FUNCTION_BLOCK ItpResetFastMFuncEx
VAR_INPUT
	bExecute:	BOOL;
	nMFuncNo:	UINT;
	tTimeOut:	TIME := DEFAULT_ADS_TIMEOUT;
END_VAR
VAR_IN_OUT
	sNciToPlc:	NciChannelToPlc;
END_VAR
VAR_OUTPUT
	bBusy:	BOOL	:= FALSE;
	bErr:		BOOL	:= FALSE;
	nErrId:	UDINT	:= 0;
END_VAR
VAR
	nState:		UDINT := 0;
	fbItpResetFastMFunc:	ItpResetFastMFunc;
END_VAR
CASE nState OF
0:
	IF bExecute THEN
		IF ItpGetItfVersion( sNciToPlc ) > 0 THEN
			fbItpResetFastMFunc(
				bExecute	:= TRUE,
				nChnId	:= ItpGetChannelId( sNciToPlc ),
				nMFuncNo	:= nMFuncNo,
				tTimeOut:= tTimeOut,
				bBusy	=> bBusy,
				bErr	=> bErr,
				nErrId=> nErrId );
			nState	:= 10;
		ELSE
			bBusy		:= TRUE;
			bErr		:= TRUE;
			nErrId	:= ErrTcNciItp_ItfVersion;
			nState	:= 9999;
		END_IF
	END_IF
10:
	fbItpResetFastMFunc();
	IF NOT fbItpResetFastMFunc.bBusy THEN
		bBusy	:= FALSE;
		IF NOT fbItpResetFastMFunc.bErr THEN
			IF NOT bExecute THEN
				fbItpResetFastMFunc( bExecute := FALSE );
				nState	:= 0;
			ELSE
				nState	:= 9999;
			END_IF
		ELSE
			bErr		:= TRUE;
			nErrId	:= fbItpResetFastMFunc.nErrId;
			nState	:= 9999;
		END_IF
	END_IF

9999:
	fbItpResetFastMFunc( bExecute:=FALSE );
	bBusy	:= FALSE;
	IF NOT bExecute THEN
		nState	:= 0;
	END_IF

END_CASE
END_FUNCTION_BLOCK

(* POU ItpRetraceMoveBackward, ST *)
(*==========================================================*)
(* Name:			ItpRetraceMoveBackward  							*)
(* Desc:			THIS IS NOT A RELEASED IMPLEMENTATION AND    *)
(*             SUBJECT TO CHANGE                            *)
(*             Moving backward                              *)
(*             - program stopped with ItpEStop              *)
(*             - FeederBackup must be enabled               *)
(* Author:	 	kbn														*)
(* Date:			07-december-2006										*)
(* last edit:	VER 6.2.33 						                  *)
(*==========================================================*)
FUNCTION_BLOCK ItpRetraceMoveBackward
VAR_INPUT
	bExecute:	BOOL;
	tTimeOut:	TIME := DEFAULT_ADS_TIMEOUT;
END_VAR
VAR_IN_OUT
	sNciToPlc:	NciChannelToPlc;
END_VAR
VAR_OUTPUT
	bBusy:		BOOL	:= FALSE;
	bErr:			BOOL	:= FALSE;
	nErrId:		UDINT	:= 0;
END_VAR
VAR
	nState:		UDINT	:= 0;
	nData:		UDINT	:= 0;
	fbAdsWrite:	ADSWRITE;
	tDummy:		ST_ItpRetrace;
	fbIsBackupEnabled:ItpIsFeederBackupEnabled;
END_VAR
CASE nState OF
0:
	IF bExecute THEN
		IF ItpGetItfVersion( sNciToPlc ) >= 3 THEN
			bBusy		:= TRUE;
			bErr		:= FALSE;
			nErrId	:= 0;
			nState	:= 10;
		ELSE
			bBusy		:= TRUE;
			bErr		:= TRUE;
			nErrId	:= ErrTcNciItp_ItfVersion;
			nState	:= 9999;
		END_IF
	END_IF
10:
	(* check, if backup is enabled *)
	fbIsBackupEnabled(
		bExecute	:= TRUE,
		tTimeOut	:= tTimeOut,
		sNciToPlc:= sNciToPlc );
	IF NOT fbIsBackupEnabled.bBusy THEN
		IF NOT fbIsBackupEnabled.bErr THEN
			IF fbIsBackupEnabled.bEnabled THEN
				nState	:= 15;
			ELSE
				(* not enabled - fire an error *)
				bErr		:= TRUE;
				nErrId	:= ErrTcNciItp_NotEnabled;
				nState	:= 9999;
			END_IF
		ELSE
			bErr		:= TRUE;
			nErrId	:= fbIsBackupEnabled.nErrId;
			nState	:= 9999;
		END_IF
		fbIsBackupEnabled( bExecute := FALSE, sNciToPlc:= sNciToPlc );
	END_IF

15:
	(* add some code to ensure, that axes stand still *)
	(* in the moment I just check, if e-stop is active *)
	IF NOT ItpIsEStopEx( sNciToPlc ) THEN
		bErr		:= TRUE;
		nErrId	:= ErrTcNciItp_NotReady;
		nState	:= 9999;
	ELSE
		fbAdsWrite(
			NETID		:= '',
			PORT		:= g_NcPortTcNci,
			IDXGRP	:= NCIDXG_CHNFUNCS + ItpGetChannelId(sNciToPlc:=sNciToPlc),
			IDXOFFS	:= 16#14,
			LEN		:= SIZEOF( tDummy ),
			SRCADDR	:= ADR( tDummy ),
			WRITE		:= TRUE,
			TMOUT		:= tTimeOut );
		nState	:= 20;
	END_IF

20:
	fbAdsWrite();
	IF NOT fbAdsWrite.BUSY THEN
		IF NOT fbAdsWrite.ERR THEN
			IF NOT bExecute THEN
				fbAdsWrite( WRITE := FALSE );
				nState	:= 0;
			ELSE
				nState	:= 9999;
			END_IF
			bBusy	:= FALSE;
		ELSE
			bErr		:= TRUE;
			nErrId	:= fbAdsWrite.ERRID;
			nState	:= 9999;
		END_IF
	END_IF

9999:
	bBusy	:= FALSE;
	fbAdsWrite( WRITE := FALSE );
	IF NOT bExecute THEN
		nState	:= 0;
	END_IF

END_CASE
END_FUNCTION_BLOCK

(* POU ItpRetraceMoveForward, ST *)
(*==========================================================*)
(* Name:			ItpRetraceMoveForward    							*)
(* Desc:			THIS IS NOT A RELEASED IMPLEMENTATION AND    *)
(*             SUBJECT TO CHANGE                            *)
(*             Moving forward again after retrace           *)
(*             - program stopped with ItpEStop              *)
(*             - FeederBackup must be enabled               *)
(* Author:	 	kbn														*)
(* Date:			07-december-2006										*)
(* last edit:	VER 6.2.33 						                  *)
(*==========================================================*)
FUNCTION_BLOCK ItpRetraceMoveForward
VAR_INPUT
	bExecute:	BOOL;
	tTimeOut:	TIME := DEFAULT_ADS_TIMEOUT;
END_VAR
VAR_IN_OUT
	sNciToPlc:	NciChannelToPlc;
END_VAR
VAR_OUTPUT
	bBusy:		BOOL	:= FALSE;
	bErr:			BOOL	:= FALSE;
	nErrId:		UDINT	:= 0;
END_VAR
VAR
	nState:		UDINT	:= 0;
	nData:		UDINT	:= 0;
	fbAdsWrite:	ADSWRITE;
	tDummy:		ST_ItpRetrace;
	fbIsBackupEnabled:ItpIsFeederBackupEnabled;
END_VAR
CASE nState OF
0:
	IF bExecute THEN
		IF ItpGetItfVersion( sNciToPlc ) >= 3 THEN
			bBusy		:= TRUE;
			bErr		:= FALSE;
			nErrId	:= 0;
			nState	:= 10;
		ELSE
			bBusy		:= TRUE;
			bErr		:= TRUE;
			nErrId	:= ErrTcNciItp_ItfVersion;
			nState	:= 9999;
		END_IF
	END_IF
10:
	(* check, if backup is enabled *)
	fbIsBackupEnabled(
		bExecute	:= TRUE,
		tTimeOut	:= tTimeOut,
		sNciToPlc:= sNciToPlc );
	IF NOT fbIsBackupEnabled.bBusy THEN
		IF NOT fbIsBackupEnabled.bErr THEN
			IF fbIsBackupEnabled.bEnabled THEN
				nState	:= 15;
			ELSE
				(* not enabled - fire an error *)
				bErr		:= TRUE;
				nErrId	:= ErrTcNciItp_NotEnabled;
				nState	:= 9999;
			END_IF
		ELSE
			bErr		:= TRUE;
			nErrId	:= fbIsBackupEnabled.nErrId;
			nState	:= 9999;
		END_IF
		fbIsBackupEnabled( bExecute := FALSE, sNciToPlc:= sNciToPlc );
	END_IF
15:
	(* add some code to ensure, that axes stand still *)
	(* in the moment I just check, if e-stop is active *)
	IF NOT ItpIsEStopEx( sNciToPlc ) THEN
		bErr		:= TRUE;
		nErrId	:= ErrTcNciItp_NotReady;
		nState	:= 9999;
	ELSE
		fbAdsWrite(
			NETID		:= '',
			PORT		:= g_NcPortTcNci,
			IDXGRP	:= NCIDXG_CHNFUNCS + ItpGetChannelId(sNciToPlc:=sNciToPlc),
			IDXOFFS	:= 16#15,
			LEN		:= SIZEOF( tDummy ),
			SRCADDR	:= ADR( tDummy ),
			WRITE		:= TRUE,
			TMOUT		:= tTimeOut );
		nState	:= 20;
	END_IF

20:
	fbAdsWrite();
	IF NOT fbAdsWrite.BUSY THEN
		IF NOT fbAdsWrite.ERR THEN
			IF NOT bExecute THEN
				fbAdsWrite( WRITE := FALSE );
				nState	:= 0;
			ELSE
				nState	:= 9999;
			END_IF
			bBusy	:= FALSE;
		ELSE
			bErr		:= TRUE;
			nErrId	:= fbAdsWrite.ERRID;
			nState	:= 9999;
		END_IF
	END_IF

9999:
	bBusy	:= FALSE;
	fbAdsWrite( WRITE := FALSE );
	IF NOT bExecute THEN
		nState	:= 0;
	END_IF

END_CASE
END_FUNCTION_BLOCK

(* POU ItpSetBottleNeckLookAhead, ST *)
(* Name:			ItpSetBottleNeckLookAhead  						*)
(* Desc:			sets the size of the look ahead for the 		*)
(*             contour collision detection (bottle neck)    *)
(* Author:	 	kbn														*)
(* Date:			26-March-2002											*)
(* Revision:	VER 5.3.4  												*)
(* last edit:	VER 6.2.33 						                  *)
(*==========================================================*)

FUNCTION_BLOCK ItpSetBottleNeckLookAhead
VAR_INPUT
	bExecute:	BOOL;
	nChnId:		UDINT;
	nLookAhead:	UDINT;
	tTimeOut:	TIME := DEFAULT_ADS_TIMEOUT;
END_VAR
VAR_OUTPUT
	bBusy:	BOOL	:= FALSE;
	bErr:		BOOL	:= FALSE;
	nErrId:	UDINT	:= 0;
END_VAR
VAR
	nState:		UDINT	:= 0;
	fbAdsWrite:	ADSWRITE;
END_VAR
VAR CONSTANT
	IDXO_CHNP_BNLOOKAHEAD:	UDINT	:= 16#51;
END_VAR
(*
Version history:
09/22/2003    | 5.4.13     | V2.9.0 (Build 947) | kbn             | adjustable target port cf. issue #2304
              |            | saved as 2.8       |                 |
*)
CASE nState OF

0:
	(* wait on trigger event *)
	IF bExecute THEN
		bBusy		:= TRUE;
		bErr		:= FALSE;
		nErrId	:= 0;

		fbAdsWrite(
			NETID		:= '',
			PORT		:= g_NcPortTcNci,
			IDXGRP	:= NCIDXG_CHN_PARMS + nChnId,
			IDXOFFS	:= IDXO_CHNP_BNLOOKAHEAD,
			LEN		:= SIZEOF( nLookAhead ),
			SRCADDR	:= ADR( nLookAhead ),
			WRITE		:= TRUE,
			TMOUT		:= tTimeOut );

		nState	:= 10;
	END_IF

10:
	fbAdsWrite();

	IF NOT fbAdsWrite.BUSY THEN
		IF NOT fbAdsWrite.ERR THEN
			IF NOT bExecute THEN
				fbAdsWrite( WRITE := FALSE );
				nState	:= 0;
			ELSE
				nState	:= 20;
			END_IF
			bBusy	:= FALSE;
		ELSE
			bErr		:= TRUE;
			nErrId	:= fbAdsWrite.ERRID;
			nState	:= 20;
		END_IF
	END_IF

20:
	fbAdsWrite( WRITE := FALSE );
	bBusy	:= FALSE;

	IF NOT bExecute THEN
		nState	:= 0;
	END_IF

END_CASE
END_FUNCTION_BLOCK

(* POU ItpSetBottleNeckLookAheadEx, ST *)
(*==========================================================*)
(* Name:			ItpSetBottleNeckLookAheadEx						*)
(* Desc:       sets the size of the look ahead for the 		*)
(*             contour collision detection (bottle neck)    *)
(* Author:	 	kbn														*)
(* Date:			26-September-2006										*)
(* last edit:	VER 6.2.33 						                  *)
(*==========================================================*)

FUNCTION_BLOCK ItpSetBottleNeckLookAheadEx
VAR_INPUT
	bExecute:	BOOL;
	nLookAhead:	UDINT;
	tTimeOut:	TIME := DEFAULT_ADS_TIMEOUT;
END_VAR
VAR_IN_OUT
	sNciToPlc:	NciChannelToPlc;
END_VAR
VAR_OUTPUT
	bBusy:	BOOL	:= FALSE;
	bErr:		BOOL	:= FALSE;
	nErrId:	UDINT	:= 0;
END_VAR
VAR
	nState:		UDINT := 0;
	fbSetBottleNeckNookAhead:	ItpSetBottleNeckLookAhead;
END_VAR
CASE nState OF
0:
	IF bExecute THEN
		IF ItpGetItfVersion( sNciToPlc ) > 0 THEN
			fbSetBottleNeckNookAhead(
				bExecute	:= TRUE,
				nChnId	:= ItpGetChannelId( sNciToPlc ),
				nLookAhead:= nLookAhead,
				tTimeOut	:= tTimeOut,
				bBusy	=> bBusy,
				bErr	=> bErr,
				nErrId=> nErrId );
			nState	:= 10;
		ELSE
			bBusy		:= TRUE;
			bErr		:= TRUE;
			nErrId	:= ErrTcNciItp_ItfVersion;
			nState	:= 9999;
		END_IF
	END_IF
10:
	fbSetBottleNeckNookAhead();
	IF NOT fbSetBottleNeckNookAhead.bBusy THEN
		bBusy	:= FALSE;
		IF NOT fbSetBottleNeckNookAhead.bErr THEN
			IF NOT bExecute THEN
				fbSetBottleNeckNookAhead( bExecute := FALSE );
				nState	:= 0;
			ELSE
				nState	:= 9999;
			END_IF
		ELSE
			bErr		:= TRUE;
			nErrId	:= fbSetBottleNeckNookAhead.nErrId;
			nState	:= 9999;
		END_IF
	END_IF

9999:
	fbSetBottleNeckNookAhead( bExecute:=FALSE );
	bBusy	:= FALSE;
	IF NOT bExecute THEN
		nState	:= 0;
	END_IF

END_CASE
END_FUNCTION_BLOCK

(* POU ItpSetBottleNeckMode, ST *)
(* Name:			ItpSetBottleNeckMode        						*)
(* Desc:			parametrize the reaction if a contour        *)
(*             collision is detected                        *)
(* Author:	 	kbn														*)
(* Date:			26-March-2002											*)
(* Revision:	VER 5.3.4  												*)
(* last edit:	VER 6.2.33 						                  *)
(*==========================================================*)

FUNCTION_BLOCK ItpSetBottleNeckMode
VAR_INPUT
	bExecute:			BOOL;
	nChnId:				UDINT;
	eBottleNeckMode:	E_ItpBnMode;
	tTimeOut:			TIME := DEFAULT_ADS_TIMEOUT;
END_VAR
VAR_OUTPUT
	bBusy:	BOOL	:= FALSE;
	bErr:		BOOL	:= FALSE;
	nErrId:	UDINT	:= 0;
END_VAR
VAR
	nState:		UDINT	:= 0;
	fbAdsWrite:	ADSWRITE;
	nTemp:		UDINT;
END_VAR
VAR CONSTANT
	IDXO_CHNP_BNMODE:	UDINT	:= 16#50;
END_VAR
(*
Version history:
09/22/2003    | 5.4.13     | V2.9.0 (Build 947) | kbn             | adjustable target port cf. issue #2304
              |            | saved as 2.8       |                 |
*)
CASE nState OF

0:
	(* wait on trigger event *)
	IF bExecute THEN
		bBusy		:= TRUE;
		bErr		:= FALSE;
		nErrId	:= 0;

		nTemp	:= INT_TO_UDINT( eBottleNeckMode );

		fbAdsWrite(
			NETID		:= '',
			PORT		:= g_NcPortTcNci,
			IDXGRP	:= NCIDXG_CHN_PARMS + nChnId,
			IDXOFFS	:= IDXO_CHNP_BNMODE,
			LEN		:= SIZEOF( nTemp ),
			SRCADDR	:= ADR( nTemp ),
			WRITE		:= TRUE,
			TMOUT		:= tTimeOut );

		nState	:= 10;
	END_IF

10:
	fbAdsWrite();

	IF NOT fbAdsWrite.BUSY THEN
		IF NOT fbAdsWrite.ERR THEN
			IF NOT bExecute THEN
				fbAdsWrite( WRITE := FALSE );
				nState	:= 0;
			ELSE
				nState	:= 20;
			END_IF
			bBusy	:= FALSE;
		ELSE
			bErr		:= TRUE;
			nErrId	:= fbAdsWrite.ERRID;
			nState	:= 20;
		END_IF
	END_IF

20:
	fbAdsWrite( WRITE := FALSE );
	bBusy	:= FALSE;

	IF NOT bExecute THEN
		nState	:= 0;
	END_IF

END_CASE
END_FUNCTION_BLOCK

(* POU ItpSetBottleNeckModeEx, ST *)
(*==========================================================*)
(* Name:			ItpSetBottleNeckModeEx								*)
(* Desc:		   parametrize the reaction if a contour        *)
(*             collision is detected                        *)
(* Author:	 	kbn														*)
(* Date:			26-September-2006										*)
(* last edit:	VER 6.2.33 						                  *)
(*==========================================================*)

FUNCTION_BLOCK ItpSetBottleNeckModeEx
VAR_INPUT
	bExecute:			BOOL;
	eBottleNeckMode:	E_ItpBnMode;
	tTimeOut:			TIME := DEFAULT_ADS_TIMEOUT;
END_VAR
VAR_IN_OUT
	sNciToPlc:	NciChannelToPlc;
END_VAR
VAR_OUTPUT
	bBusy:	BOOL	:= FALSE;
	bErr:		BOOL	:= FALSE;
	nErrId:	UDINT	:= 0;
END_VAR
VAR
	nState:		UDINT := 0;
	fbSetBottleNeckMode:	ItpSetBottleNeckMode;
END_VAR
CASE nState OF
0:
	IF bExecute THEN
		IF ItpGetItfVersion( sNciToPlc ) > 0 THEN
			fbSetBottleNeckMode(
				bExecute	:= TRUE,
				nChnId	:= ItpGetChannelId( sNciToPlc ),
				eBottleNeckMode	:= eBottleNeckMode,
				tTimeOut	:= tTimeOut,
				bBusy	=> bBusy,
				bErr	=> bErr,
				nErrId=> nErrId );
			nState	:= 10;
		ELSE
			bBusy		:= TRUE;
			bErr		:= TRUE;
			nErrId	:= ErrTcNciItp_ItfVersion;
			nState	:= 9999;
		END_IF
	END_IF
10:
	fbSetBottleNeckMode();
	IF NOT fbSetBottleNeckMode.bBusy THEN
		bBusy	:= FALSE;
		IF NOT fbSetBottleNeckMode.bErr THEN
			IF NOT bExecute THEN
				fbSetBottleNeckMode( bExecute := FALSE );
				nState	:= 0;
			ELSE
				nState	:= 9999;
			END_IF
		ELSE
			bErr		:= TRUE;
			nErrId	:= fbSetBottleNeckMode.nErrId;
			nState	:= 9999;
		END_IF
	END_IF

9999:
	fbSetBottleNeckMode( bExecute:=FALSE );
	bBusy	:= FALSE;
	IF NOT bExecute THEN
		nState	:= 0;
	END_IF

END_CASE
END_FUNCTION_BLOCK

(* POU ItpSetCyclicLRealOffsets, ST *)
(*==========================================================*)
(* Name:			ItpSetCyclicLRealOffsets							*)
(* Desc:			THIS IS NOT A RELEASED IMPLEMENTATION AND    *)
(*             SUBJECT TO CHANGE                            *)
(*             specifies index offsets for cylcic channel   *)
(*             interface                                    *)
(* Author:	 	kbn														*)
(* Date:			08-October-2007										*)
(* last edit:	VER 6.2.33 						                  *)
(*==========================================================*)
FUNCTION_BLOCK ItpSetCyclicLRealOffsets
VAR_INPUT
	bExecute:	BOOL;
	tTimeOut:	TIME := DEFAULT_ADS_TIMEOUT;
	nIndexOffsetParam1:	UDINT := 0;
	nIndexOffsetParam2:	UDINT := 0;
	nIndexOffsetParam3:	UDINT := 0;
	nIndexOffsetParam4:	UDINT := 0;
END_VAR
VAR_IN_OUT
	sNciToPlc:	NciChannelToPlc;
END_VAR
VAR_OUTPUT
	bBusy:		BOOL	:= FALSE;
	bErr:			BOOL	:= FALSE;
	nErrId:		UDINT	:= 0;
END_VAR
VAR
	nState:	UDINT	:= 0;
	nIndexOffsets: ARRAY[1..4] OF UDINT;
	fbAdsWrite:		ADSWRITE;
END_VAR
CASE nState OF
0:
	IF  bExecute THEN
		bBusy	:= TRUE;
		bErr	:= FALSE;
		nErrId	:= 0;

		nIndexOffsets[1]	:= nIndexOffsetParam1;
		nIndexOffsets[2]	:= nIndexOffsetParam2;
		nIndexOffsets[3]	:= nIndexOffsetParam3;
		nIndexOffsets[4]	:= nIndexOffsetParam4;

		fbAdsWrite(
			NETID		:= '',
			PORT		:= g_NcPortTcNci,
			IDXGRP	:= NCIDXG_CHNPARMS + ItpGetChannelId(sNciToPlc:=sNciToPlc),
			IDXOFFS	:= 16#56,
			LEN		:= SIZEOF(nIndexOffsets),
			SRCADDR	:= ADR(nIndexOffsets),
			WRITE		:= TRUE,
			TMOUT		:= tTimeOut);

		nState	:= 10;
	END_IF

10:
	fbAdsWrite();

	IF NOT fbAdsWrite.BUSY THEN
		IF NOT fbAdsWrite.ERR THEN
			IF NOT bExecute THEN
				fbAdsWrite( WRITE := FALSE );
				nState	:= 0;
			ELSE
				nState	:= 20;
			END_IF
			bBusy		:= FALSE;
		ELSE
			bErr		:= TRUE;
			nErrId	:= fbAdsWrite.ERRID;
			nState	:= 20;
		END_IF
	END_IF

20:
	fbAdsWrite( WRITE:= FALSE );
	bBusy		:= FALSE;
	IF NOT bExecute THEN
		nState	:= 0;
	END_IF

END_CASE
END_FUNCTION_BLOCK

(* POU ItpSetCyclicUdintOffsets, ST *)
(*==========================================================*)
(* Name:			ItpSetCyclicUdintOffsets							*)
(* Desc:			THIS IS NOT A RELEASED IMPLEMENTATION AND    *)
(*             SUBJECT TO CHANGE                            *)
(*             specifies index offsets for cylcic channel   *)
(*             interface                                    *)
(* Author:	 	kbn														*)
(* Date:			08-October-2007										*)
(* last edit:	VER 6.2.33 						                  *)
(*==========================================================*)
FUNCTION_BLOCK ItpSetCyclicUdintOffsets
VAR_INPUT
	bExecute:	BOOL;
	tTimeOut:	TIME := DEFAULT_ADS_TIMEOUT;
	nIndexOffsetParam1:	UDINT := 0;
	nIndexOffsetParam2:	UDINT := 0;
	nIndexOffsetParam3:	UDINT := 0;
	nIndexOffsetParam4:	UDINT := 0;
END_VAR
VAR_IN_OUT
	sNciToPlc:	NciChannelToPlc;
END_VAR
VAR_OUTPUT
	bBusy:		BOOL	:= FALSE;
	bErr:			BOOL	:= FALSE;
	nErrId:		UDINT	:= 0;
END_VAR
VAR
	nState:	UDINT	:= 0;
	nIndexOffsets: ARRAY[1..4] OF UDINT;
	fbAdsWrite:		ADSWRITE;
END_VAR
CASE nState OF
0:
	IF  bExecute THEN
		bBusy	:= TRUE;
		bErr	:= FALSE;
		nErrId	:= 0;

		nIndexOffsets[1]	:= nIndexOffsetParam1;
		nIndexOffsets[2]	:= nIndexOffsetParam2;
		nIndexOffsets[3]	:= nIndexOffsetParam3;
		nIndexOffsets[4]	:= nIndexOffsetParam4;

		fbAdsWrite(
			NETID		:= '',
			PORT		:= g_NcPortTcNci,
			IDXGRP	:= NCIDXG_CHNPARMS + ItpGetChannelId(sNciToPlc:=sNciToPlc),
			IDXOFFS	:= 16#55,
			LEN		:= SIZEOF(nIndexOffsets),
			SRCADDR	:= ADR(nIndexOffsets),
			WRITE		:= TRUE,
			TMOUT		:= tTimeOut);

		nState	:= 10;
	END_IF

10:
	fbAdsWrite();

	IF NOT fbAdsWrite.BUSY THEN
		IF NOT fbAdsWrite.ERR THEN
			IF NOT bExecute THEN
				fbAdsWrite( WRITE := FALSE );
				nState	:= 0;
			ELSE
				nState	:= 20;
			END_IF
			bBusy		:= FALSE;
		ELSE
			bErr		:= TRUE;
			nErrId	:= fbAdsWrite.ERRID;
			nState	:= 20;
		END_IF
	END_IF

20:
	fbAdsWrite( WRITE:= FALSE );
	bBusy		:= FALSE;
	IF NOT bExecute THEN
		nState	:= 0;
	END_IF

END_CASE
END_FUNCTION_BLOCK

(* POU ItpSetOverridePercent, ST *)
(* Name:			ItpSetOverridePercent								*)
(* Desc:			sets the override in the cyclic interface		*)
(* Author:	 	kbn														*)
(* Date:			30-May-2001												*)
(* Revision:	VER 4.0.0  												*)
(*==========================================================*)

FUNCTION ItpSetOverridePercent : BOOL
VAR_IN_OUT
	sPlcToNci:	NciChannelFromPlc;
END_VAR
VAR_INPUT
	fOverridePercent:	LREAL;
END_VAR
VAR
END_VAR
sPlcToNci.nChaAxesOvr	:= LREAL_TO_DWORD( fOverridePercent * 10000.0 );
ItpSetOverridePercent 	:= TRUE;
END_FUNCTION

(* POU ItpSetSubroutinePath, ST *)
(*==========================================================*)
(* Name:			ItpSetSubroutinePath									*)
(* Desc:			sets search path for subroutines					*)
(* Author:	 	kbn														*)
(* Date:			24-June-2004											*)
(* Revision:	VER 5.4.17 	#2578										*)
(* last edit:	VER 6.2.33 						                  *)
(*==========================================================*)

FUNCTION_BLOCK ItpSetSubroutinePath
VAR_INPUT
	bExecute:	BOOL;
	nChnId:		UDINT;
	sPath:		STRING;
	nLength:		UDINT;
	tTimeOut:	TIME := DEFAULT_ADS_TIMEOUT;
END_VAR
VAR_OUTPUT
	bBusy:	BOOL	:= FALSE;
	bErr:		BOOL	:= FALSE;
	nErrId:	UDINT	:= 0;
END_VAR
VAR
	nState:		UDINT	:= 0;
	fbAdsWrite:	ADSWRITE;
END_VAR
CASE nState OF

0:
	(* wait on trigger event *)
	IF bExecute THEN
		bBusy	:= TRUE;
		bErr	:= FALSE;
		nErrId	:= 0;

		fbAdsWrite(
			NETID		:= '',
			PORT		:= g_NcPortTcNci,
			IDXGRP	:= NCIDXG_CHN_FUNCS + nChnId,
			IDXOFFS	:= 6,
			LEN		:= nLength,
			SRCADDR	:= ADR(sPath),
			WRITE		:= TRUE,
			TMOUT		:= tTimeOut);

		nState	:= 10;
	END_IF

10:
	(* execute AdsWrite command *)
	fbAdsWrite();

	IF NOT fbAdsWrite.BUSY THEN
		IF NOT fbAdsWrite.ERR THEN
			IF NOT bExecute THEN
				fbAdsWrite( WRITE := FALSE );
				nState	:= 0;
			ELSE
				nState	:= 20;
			END_IF
			bBusy	:= FALSE;
		ELSE
			bErr		:= TRUE;
			nErrId	:= fbAdsWrite.ERRID;
			nState	:= 20;
		END_IF
	END_IF
20:
	fbAdsWrite( WRITE := FALSE );
	bBusy	:= FALSE;
	IF NOT bExecute THEN
		nState	:= 0;
	END_IF
END_CASE
END_FUNCTION_BLOCK

(* POU ItpSetSubroutinePathEx, ST *)
(*==========================================================*)
(* Name:			ItpSetSubroutinePathEx 								*)
(* Desc:			sets search path for subroutines					*)
(* Author:	 	kbn														*)
(* Date:			26-September-2006										*)
(* last edit:	VER 6.2.33 						                  *)
(*==========================================================*)

FUNCTION_BLOCK ItpSetSubroutinePathEx
VAR_INPUT
	bExecute:	BOOL;
	sPath:		STRING;
	nLength:		UDINT;
	tTimeOut:	TIME := DEFAULT_ADS_TIMEOUT;
END_VAR
VAR_IN_OUT
	sNciToPlc:	NciChannelToPlc;
END_VAR
VAR_OUTPUT
	bBusy:	BOOL	:= FALSE;
	bErr:		BOOL	:= FALSE;
	nErrId:	UDINT	:= 0;
END_VAR
VAR
	nState:		UDINT := 0;
	fbItpSetSubroutinePath:	ItpSetSubroutinePath;
END_VAR
(*
	nChnId:		UDINT;
*)

CASE nState OF
0:
	IF bExecute THEN
		IF ItpGetItfVersion( sNciToPlc ) > 0 THEN
			fbItpSetSubroutinePath(
				bExecute	:= TRUE,
				nChnId	:= ItpGetChannelId( sNciToPlc ),
				sPath		:= sPath,
				nLength	:= nLength,
				tTimeOut:= tTimeOut,
				bBusy	=> bBusy,
				bErr	=> bErr,
				nErrId=> nErrId );
			nState	:= 10;
		ELSE
			bBusy		:= TRUE;
			bErr		:= TRUE;
			nErrId	:= ErrTcNciItp_ItfVersion;
			nState	:= 9999;
		END_IF
	END_IF
10:
	fbItpSetSubroutinePath();
	IF NOT fbItpSetSubroutinePath.bBusy THEN
		bBusy	:= FALSE;
		IF NOT fbItpSetSubroutinePath.bErr THEN
			IF NOT bExecute THEN
				fbItpSetSubroutinePath( bExecute := FALSE );
				nState	:= 0;
			ELSE
				nState	:= 9999;
			END_IF
		ELSE
			bErr		:= TRUE;
			nErrId	:= fbItpSetSubroutinePath.nErrId;
			nState	:= 9999;
		END_IF
	END_IF

9999:
	fbItpSetSubroutinePath( bExecute:=FALSE );
	bBusy	:= FALSE;
	IF NOT bExecute THEN
		nState	:= 0;
	END_IF

END_CASE
END_FUNCTION_BLOCK

(* POU ItpSetToolDescNull, ST *)
(*==========================================================*)
(* ItpSetToolDescNull													*)
(* Desc:			set all tool descriptions to null            *)
(* Author:	 	kbn														*)
(* Date:			17-June-2005											*)
(* Revision:	VER 5.5.18 												*)
(* last edit:	VER 6.2.33 						                  *)
(*==========================================================*)

FUNCTION_BLOCK ItpSetToolDescNull
VAR_INPUT
	bExecute:	BOOL;
	nChnId:		UDINT;
	tTimeOut:	TIME := DEFAULT_ADS_TIMEOUT;
END_VAR
VAR_OUTPUT
	bBusy:		BOOL	:= FALSE;
	bErr:			BOOL	:= FALSE;
	nErrId:		UDINT	:= 0;
END_VAR
VAR
	nState:		UDINT	:= 0;
	fbAdsWrite:	ADSWRITE;
END_VAR
CASE nState OF

0:
	(* wait on trigger event *)
	IF bExecute THEN
		bBusy	:= TRUE;
		bErr	:= FALSE;
		nErrId	:= 0;

		fbAdsWrite(
			NETID		:= '',
			PORT		:= g_NcPortTcNci,
			IDXGRP	:= NCIDXG_CHN_FUNCS + nChnId,
			IDXOFFS	:= 16#26,
			LEN		:= 0,
			SRCADDR	:= 0,
			WRITE		:= TRUE,
			TMOUT		:= tTimeOut);

		nState	:= 10;
	END_IF

10:
	(* execute  command *)
	fbAdsWrite();

	IF NOT fbAdsWrite.BUSY THEN
		IF NOT fbAdsWrite.ERR THEN
			IF NOT bExecute THEN
				fbAdsWrite( WRITE := FALSE );
				nState	:= 0;
			ELSE
				nState	:= 20;
			END_IF
			bBusy	:= FALSE;
		ELSE
			bErr		:= TRUE;
			nErrId	:= fbAdsWrite.ERRID;
			nState	:= 20;
		END_IF
	END_IF
20:
	fbAdsWrite( WRITE := FALSE );
	bBusy	:= FALSE;
	IF NOT bExecute THEN
		nState	:= 0;
	END_IF
END_CASE
END_FUNCTION_BLOCK

(* POU ItpSetToolDescNullEx, ST *)
(*==========================================================*)
(* Name:			ItpSetToolDescNullEx								   *)
(* Desc:		   set all tool descriptions to null            *)
(* Author:	 	kbn														*)
(* Date:			26-September-2006										*)
(* last edit:	VER 6.2.33 						                  *)
(*==========================================================*)

FUNCTION_BLOCK ItpSetToolDescNullEx
VAR_INPUT
	bExecute:	BOOL;
	tTimeOut:	TIME := DEFAULT_ADS_TIMEOUT;
END_VAR
VAR_IN_OUT
	sNciToPlc:	NciChannelToPlc;
END_VAR
VAR_OUTPUT
	bBusy:	BOOL	:= FALSE;
	bErr:		BOOL	:= FALSE;
	nErrId:	UDINT	:= 0;
END_VAR
VAR
	nState:		UDINT := 0;
	fbSetToolDescNull:	ItpSetToolDescNull;
END_VAR
CASE nState OF
0:
	IF bExecute THEN
		IF ItpGetItfVersion( sNciToPlc ) > 0 THEN
			fbSetToolDescNull(
				bExecute	:= TRUE,
				nChnId	:= ItpGetChannelId( sNciToPlc ),
				tTimeOut	:= tTimeOut,
				bBusy	=> bBusy,
				bErr	=> bErr,
				nErrId=> nErrId );
			nState	:= 10;
		ELSE
			bBusy		:= TRUE;
			bErr		:= TRUE;
			nErrId	:= ErrTcNciItp_ItfVersion;
			nState	:= 9999;
		END_IF
	END_IF
10:
	fbSetToolDescNull();
	IF NOT fbSetToolDescNull.bBusy THEN
		bBusy	:= FALSE;
		IF NOT fbSetToolDescNull.bErr THEN
			IF NOT bExecute THEN
				fbSetToolDescNull( bExecute := FALSE );
				nState	:= 0;
			ELSE
				nState	:= 9999;
			END_IF
		ELSE
			bErr		:= TRUE;
			nErrId	:= fbSetToolDescNull.nErrId;
			nState	:= 9999;
		END_IF
	END_IF

9999:
	fbSetToolDescNull( bExecute:=FALSE );
	bBusy	:= FALSE;
	IF NOT bExecute THEN
		nState	:= 0;
	END_IF

END_CASE
END_FUNCTION_BLOCK

(* POU ItpSetZeroShiftNull, ST *)
(*==========================================================*)
(* ItpSetZeroShiftNull													*)
(* Desc:			set all zero shifts to null                  *)
(* Author:	 	kbn														*)
(* Date:			17-June-2005											*)
(* Revision:	VER 5.5.18 												*)
(* last edit:	VER 6.2.33 						                  *)
(*==========================================================*)

FUNCTION_BLOCK ItpSetZeroShiftNull
VAR_INPUT
	bExecute:	BOOL;
	nChnId:		UDINT;
	tTimeOut:	TIME := DEFAULT_ADS_TIMEOUT;
END_VAR
VAR_OUTPUT
	bBusy:		BOOL	:= FALSE;
	bErr:			BOOL	:= FALSE;
	nErrId:		UDINT	:= 0;
END_VAR
VAR
	nState:		UDINT	:= 0;
	fbAdsWrite:	ADSWRITE;
END_VAR
CASE nState OF

0:
	(* wait on trigger event *)
	IF bExecute THEN
		bBusy	:= TRUE;
		bErr	:= FALSE;
		nErrId	:= 0;

		fbAdsWrite(
			NETID		:= '',
			PORT		:= g_NcPortTcNci,
			IDXGRP	:= NCIDXG_CHN_FUNCS + nChnId,
			IDXOFFS	:= 16#27,
			LEN		:= 0,
			SRCADDR	:= 0,
			WRITE		:= TRUE,
			TMOUT		:= tTimeOut);

		nState	:= 10;
	END_IF

10:
	(* execute  command *)
	fbAdsWrite();

	IF NOT fbAdsWrite.BUSY THEN
		IF NOT fbAdsWrite.ERR THEN
			IF NOT bExecute THEN
				fbAdsWrite( WRITE := FALSE );
				nState	:= 0;
			ELSE
				nState	:= 20;
			END_IF
			bBusy	:= FALSE;
		ELSE
			bErr		:= TRUE;
			nErrId	:= fbAdsWrite.ERRID;
			nState	:= 20;
		END_IF
	END_IF
20:
	fbAdsWrite( WRITE := FALSE );
	bBusy	:= FALSE;
	IF NOT bExecute THEN
		nState	:= 0;
	END_IF
END_CASE
END_FUNCTION_BLOCK

(* POU ItpSetZeroShiftNullEx, ST *)
(*==========================================================*)
(* Name:			ItpSetZeroShiftNullEx							   *)
(* Desc:			set all zero shifts to null                  *)
(* Author:	 	kbn														*)
(* Date:			26-September-2006										*)
(* last edit:	VER 6.2.33 						                  *)
(*==========================================================*)

FUNCTION_BLOCK ItpSetZeroShiftNullEx
VAR_INPUT
	bExecute:	BOOL;
	tTimeOut:	TIME := DEFAULT_ADS_TIMEOUT;
END_VAR
VAR_IN_OUT
	sNciToPlc:	NciChannelToPlc;
END_VAR
VAR_OUTPUT
	bBusy:		BOOL;
	bErr:			BOOL;
	nErrId:		UDINT;
END_VAR
VAR
	nState:		UDINT := 0;
	fbSetZeroShiftNull:	ItpSetZeroShiftNull;
END_VAR
CASE nState OF
0:
	IF bExecute THEN
		IF ItpGetItfVersion( sNciToPlc ) > 0 THEN
			fbSetZeroShiftNull(
				bExecute	:= TRUE,
				nChnId	:= ItpGetChannelId( sNciToPlc ),
				tTimeOut	:= tTimeOut,
				bBusy	=> bBusy,
				bErr	=> bErr,
				nErrId=> nErrId );
			nState	:= 10;
		ELSE
			bBusy		:= TRUE;
			bErr		:= TRUE;
			nErrId	:= ErrTcNciItp_ItfVersion;
			nState	:= 9999;
		END_IF
	END_IF
10:
	fbSetZeroShiftNull();
	IF NOT fbSetZeroShiftNull.bBusy THEN
		bBusy	:= FALSE;
		IF NOT fbSetZeroShiftNull.bErr THEN
			IF NOT bExecute THEN
				fbSetZeroShiftNull( bExecute := FALSE );
				nState	:= 0;
			ELSE
				nState	:= 9999;
			END_IF
		ELSE
			bErr		:= TRUE;
			nErrId	:= fbSetZeroShiftNull.nErrId;
			nState	:= 9999;
		END_IF
	END_IF

9999:
	fbSetZeroShiftNull( bExecute:=FALSE );
	bBusy	:= FALSE;
	IF NOT bExecute THEN
		nState	:= 0;
	END_IF

END_CASE
END_FUNCTION_BLOCK

(* POU ItpSingleBlock, ST *)
(*==========================================================*)
(* Name:			ItpSingleBlock       							   *)
(* Desc:			THIS IS NOT A RELEASED IMPLEMENTATION AND    *)
(*             SUBJECT TO CHANGE                            *)
(*     			- enables single block mode                  *)
(*             - triggers next block                        *)
(* Author:	 	kbn														*)
(* Date:			22-February-2008										*)
(* last edit:	VER 6.2.33 						                  *)
(*==========================================================*)

FUNCTION_BLOCK ItpSingleBlock
VAR_INPUT
	bExecuteModeChange:	BOOL;
	nMode: E_ItpSingleBlockMode	:= ItpSingleBlockOff;
	bTriggerNext:	BOOL	:= FALSE;
	tTimeOut:   TIME := DEFAULT_ADS_TIMEOUT;
END_VAR
VAR_IN_OUT
	sNciToPlc:	NciChannelToPlc;
END_VAR
VAR_OUTPUT
	bBusy:		BOOL	:= FALSE;
	bErr:			BOOL	:= FALSE;
	nErrId:		UDINT	:= 0;
END_VAR
VAR
	nStateMode:	UDINT	:= 0;
	nStateTrigger:	UDINT	:= 0;
	fbAdsWrite:	ADSWRITE;
	fbItpTrigger:ItpStartStopEx;
END_VAR
(* if single block is active sNciToPlc.mItpOpMode is 0x1 or 0x4000 *)
(* activation must be done via ads *)
(* trigger next must be done via ItpStartEx *)

fbAdsWrite(
	NETID		:= '',
	PORT		:= g_NcPortTcNci,
	IDXGRP	:= NCIDXG_CHN_FUNCS + ItpGetChannelId(sNciToPlc:=sNciToPlc),
	IDXOFFS	:= 16#5,
	LEN		:= SIZEOF(nMode),
	SRCADDR	:= ADR(nMode),
	WRITE		:= bExecuteModeChange,
	TMOUT		:= tTimeOut);


fbItpTrigger(
	bStart:=bTriggerNext,
	bStop:=FALSE,
	tTimeOut:=tTimeOut,
	sNciToPlc:=sNciToPlc );

IF fbAdsWrite.BUSY OR fbItpTrigger.bBusy THEN
	bBusy	:= TRUE;
ELSE
	bBusy	:= FALSE;
END_IF

IF fbAdsWrite.ERR THEN
	bErr	:= TRUE;
	nErrId	:= fbAdsWrite.ERRID;
ELSIF fbItpTrigger.bErr THEN
	bErr	:= TRUE;
	nErrId	:= fbItpTrigger.nErrId;
ELSE
	bErr	:= FALSE;
	nErrId	:= 0;
END_IF
END_FUNCTION_BLOCK

(* POU ItpStartStopEx, ST *)
(*==========================================================*)
(* Name:			ItpStartStopEx        							   *)
(* Desc:			starts/stops interpolation with g-code       *)
(* Author:	 	kbn														*)
(* Date:			26-September-2006										*)
(* last edit:	VER 6.2.33 						                  *)
(*==========================================================*)

FUNCTION_BLOCK ItpStartStopEx
VAR_INPUT
	bStart		:	BOOL;
	bStop			:	BOOL;
	tTimeOut		:	TIME := DEFAULT_ADS_TIMEOUT;
END_VAR
VAR_IN_OUT
	sNciToPlc:	NciChannelToPlc;
END_VAR
VAR_OUTPUT
	bBusy		:	BOOL	:= FALSE;
	bErr		:	BOOL	:= FALSE;
	nErrId	:	UDINT	:= 0;
END_VAR
VAR
	fbStartStop:	ItpStartStop;
END_VAR
IF ItpGetItfVersion( sNciToPlc ) > 0 THEN
	fbStartStop(
		bStart	:= bStart,
		bStop		:= bStop,
		nChnId	:= ItpGetChannelId( sNciToPlc ),
		tTimeOut	:= tTimeOut,
		bBusy	=> bBusy,
		bErr	=> bErr,
		nErrId=> nErrId );
ELSE
	bErr		:= TRUE;
	nErrId	:= ErrTcNciItp_ItfVersion;
END_IF
END_FUNCTION_BLOCK

(* POU ItpStepOnAfterEStop, ST *)
(* Name:       ItpStepOnAfterEStop                          *)
(* Desc:       trigger execution after estop                *)
(* Author:     kbn                                          *)
(* Date:       29-May-2002                                  *)
(* Revision:   VER 5.3.6                                    *)
(* last edit:	VER 6.2.33 						                  *)
(*==========================================================*)
FUNCTION_BLOCK ItpStepOnAfterEStop
VAR_INPUT
	bExecute:	BOOL;
	nGrpId:		UDINT;
	tTimeOut:	TIME := DEFAULT_ADS_TIMEOUT;
END_VAR
VAR_OUTPUT
	bBusy:	BOOL	:= FALSE;
	bErr:		BOOL	:= FALSE;
	nErrId:	UDINT	:= 0;
END_VAR
VAR
	nState:			UDINT := 0;
	fbAdsWrite:		ADSWRITE;
END_VAR

(*
Version history:
09/22/2003    | 5.4.13     | V2.9.0 (Build 947) | kbn             | adjustable target port cf. issue #2304
              |            | saved as 2.8       |                 |
*)
CASE nState OF
0:
	IF bExecute THEN
		bBusy		:= TRUE;
		bErr		:= FALSE;
		nErrId	:= 0;

		fbAdsWrite(
			NETID		:= '',
			PORT		:= AMSPORT_R0_NCSAF,
			IDXGRP	:= 16#3200 + nGrpId,
			IDXOFFS	:= 16#6,
			LEN		:= 0,
			SRCADDR	:= 0,
			WRITE		:= TRUE,
			TMOUT		:= tTimeOut );

		nState	:= 10;
	END_IF

10:
	fbAdsWrite();

	IF NOT fbAdsWrite.BUSY THEN
		IF NOT fbAdsWrite.ERR THEN
			IF NOT bExecute THEN
				fbAdsWrite( WRITE := FALSE );
				nState	:= 0;
			ELSE
				nState	:= 20;
			END_IF
			bBusy		:= FALSE;
		ELSE
			bErr		:= TRUE;
			nErrId	:= fbAdsWrite.ERRID;
			nState	:= 20;
		END_IF
	END_IF

20:
	fbAdsWrite( WRITE:= FALSE );
	bBusy		:= FALSE;
	IF NOT bExecute THEN
		nState	:= 0;
	END_IF

END_CASE
END_FUNCTION_BLOCK

(* POU ItpStepOnAfterEStopEx, ST *)
(*==========================================================*)
(* Name:			ItpStepOnAfterEStopEx							   *)
(* Desc:		   trigger execution after estop                *)
(* Author:	 	kbn														*)
(* Date:			26-September-2006										*)
(* last edit:	VER 6.2.33 						                  *)
(*==========================================================*)

FUNCTION_BLOCK ItpStepOnAfterEStopEx
VAR_INPUT
	bExecute:	BOOL;
	tTimeOut:	TIME := DEFAULT_ADS_TIMEOUT;
END_VAR
VAR_IN_OUT
	sNciToPlc:	NciChannelToPlc;
END_VAR
VAR_OUTPUT
	bBusy:	BOOL	:= FALSE;
	bErr:		BOOL	:= FALSE;
	nErrId:	UDINT	:= 0;
END_VAR
VAR
	nState:		UDINT := 0;
	fbStepOnAfterEStop:	ItpStepOnAfterEStop;
END_VAR
CASE nState OF
0:
	IF bExecute THEN
		IF ItpGetItfVersion( sNciToPlc ) > 0 THEN
			fbStepOnAfterEStop(
				bExecute	:= TRUE,
				nGrpId	:= ItpGetGroupId( sNciToPlc ),
				tTimeOut	:= tTimeOut,
				bBusy	=> bBusy,
				bErr	=> bErr,
				nErrId=> nErrId );
			nState	:= 10;
		ELSE
			bBusy		:= TRUE;
			bErr		:= TRUE;
			nErrId	:= ErrTcNciItp_ItfVersion;
			nState	:= 9999;
		END_IF
	END_IF
10:
	fbStepOnAfterEStop();
	IF NOT fbStepOnAfterEStop.bBusy THEN
		bBusy	:= FALSE;
		IF NOT fbStepOnAfterEStop.bErr THEN
			IF NOT bExecute THEN
				fbStepOnAfterEStop( bExecute := FALSE );
				nState	:= 0;
			ELSE
				nState	:= 9999;
			END_IF
		ELSE
			bErr		:= TRUE;
			nErrId	:= fbStepOnAfterEStop.nErrId;
			nState	:= 9999;
		END_IF
	END_IF

9999:
	fbStepOnAfterEStop( bExecute:=FALSE );
	bBusy	:= FALSE;
	IF NOT bExecute THEN
		nState	:= 0;
	END_IF

END_CASE
END_FUNCTION_BLOCK

(* POU ItpWriteRParams, ST *)
FUNCTION_BLOCK ItpWriteRParams
VAR_INPUT
	bExecute	:	BOOL;
	nChnId		:	UDINT;
	pAddr		:	DWORD;
	nIndex		:	DINT;
	nCount		:	DINT;
	tTimeOut		:	TIME := DEFAULT_ADS_TIMEOUT;
END_VAR
VAR_OUTPUT
	bBusy:	BOOL	:= FALSE;
	bErr:		BOOL	:= FALSE;
	nErrId:	UDINT	:= 0;
END_VAR
VAR CONSTANT
	(* NC ADS Index Offsets for CHANNEL Processdata *)
	NCIDXO_CHNP_RPARAMS				: UDINT := 16#10000000;

	(* states *)
	IDLE		:	INT := 0;
	START		:	INT := 1;
	WAIT		:	INT := 2;
	ERROR		:	INT := 10;
	QUIT		:	INT := 20;
END_VAR
VAR
	Dummy		:	LREAL;
	state 		:	INT := IDLE;

	(* instances *)
	AdsWrite1	:	ADSWRITE;
END_VAR

(*
Version history:
Date          | Version    | created under      | Author          | Remark 
---------------------------------------------------------------------------------------- 
02/01/2002    | 5.1.0      | V2.8.0 (Build 719) | kbn             | modified
              |            |                    |                 | - cycle optimization
---------------------------------------------------------------------------------------- 
09/22/2003    | 5.4.13     | V2.9.0 (Build 947) | kbn             | adjustable target port cf. issue #2304
              |            | saved as 2.8       |                 |
*) 
(* statemachine *)
CASE state OF

	IDLE:
		IF bExecute THEN
			bBusy := TRUE;
			bErr := FALSE;
			nErrId := 0;

			AdsWrite1.NETID		:= '';
			AdsWrite1.PORT		:= g_NcPortTcNci;
			AdsWrite1.IDXGRP	:= NCIDXG_CHN_IOAREA + nChnId;
			AdsWrite1.IDXOFFS	:= NCIDXO_CHNP_RPARAMS + nIndex;
			AdsWrite1.LEN		:= nCount * SIZEOF(Dummy);
			AdsWrite1.SRCADDR	:= pAddr;
			AdsWrite1.TMOUT	:= tTimeOut;

			IF ((nIndex-1) + nCount) > 999 THEN
				nErrId := ErrTcNciItp_RParamIndex;
				state := ERROR;
			ELSE
				IF AdsWrite1.WRITE OR AdsWrite1.BUSY THEN
					AdsWrite1( WRITE := FALSE );
				ELSE
					AdsWrite1( WRITE := TRUE );
					state := WAIT;
				END_IF
			END_IF
		END_IF

	WAIT:
(*		c.f. issue 1581*)
		AdsWrite1();
		IF NOT AdsWrite1.BUSY THEN
			IF NOT AdsWrite1.ERR THEN
				bBusy := FALSE;
				IF NOT bExecute THEN
					state := IDLE;
				ELSE
					state := QUIT;
				END_IF
			ELSE
				nErrId := AdsWrite1.ERRID;
				state := ERROR;
			END_IF
			AdsWrite1( WRITE := FALSE );
		END_IF

	ERROR:
		bErr := TRUE;
		bBusy := FALSE;
		IF NOT bExecute THEN
			state := IDLE;
		ELSE
			state := QUIT;
		END_IF

	QUIT:
		IF NOT bExecute THEN
			state := IDLE;
		END_IF

END_CASE
END_FUNCTION_BLOCK

(* POU ItpWriteRParamsEx, ST *)
(*==========================================================*)
(* Name:			ItpWriteRParamsEx							         *)
(* Desc:	      writes r-parameters to given channel         *)
(* Author:	 	kbn														*)
(* Date:			26-September-2006										*)
(* last edit:	VER 6.2.33 						                  *)
(*==========================================================*)

FUNCTION_BLOCK ItpWriteRParamsEx
VAR_INPUT
	bExecute:	BOOL;
	pAddr:		DWORD;
	nIndex:		DINT;
	nCount:		DINT;
	tTimeOut:	TIME := DEFAULT_ADS_TIMEOUT;
END_VAR
VAR_IN_OUT
	sNciToPlc:	NciChannelToPlc;
END_VAR
VAR_OUTPUT
	bBusy:	BOOL	:= FALSE;
	bErr:		BOOL	:= FALSE;
	nErrId:	UDINT	:= 0;
END_VAR
VAR
	nState:		UDINT := 0;
	fbWriteRParams:	ItpWriteRParams;
END_VAR
CASE nState OF
0:
	IF bExecute THEN
		IF ItpGetItfVersion( sNciToPlc ) > 0 THEN
			fbWriteRParams(
				bExecute	:= TRUE,
				nChnId	:= ItpGetChannelId( sNciToPlc ),
				pAddr		:= pAddr,
				nIndex	:= nIndex,
				nCount	:= nCount,
				tTimeOut	:= tTimeOut,
				bBusy	=> bBusy,
				bErr	=> bErr,
				nErrId=> nErrId );
			nState	:= 10;
		ELSE
			bBusy		:= TRUE;
			bErr		:= TRUE;
			nErrId	:= ErrTcNciItp_ItfVersion;
			nState	:= 9999;
		END_IF
	END_IF
10:
	fbWriteRParams();
	IF NOT fbWriteRParams.bBusy THEN
		bBusy	:= FALSE;
		IF NOT fbWriteRParams.bErr THEN
			IF NOT bExecute THEN
				fbWriteRParams( bExecute := FALSE );
				nState	:= 0;
			ELSE
				nState	:= 9999;
			END_IF
		ELSE
			bErr		:= TRUE;
			nErrId	:= fbWriteRParams.nErrId;
			nState	:= 9999;
		END_IF
	END_IF

9999:
	fbWriteRParams( bExecute:=FALSE );
	bBusy	:= FALSE;
	IF NOT bExecute THEN
		nState	:= 0;
	END_IF

END_CASE
END_FUNCTION_BLOCK

(* POU ItpWriteToolDesc, ST *)
(* Name:			ItpWriteToolDesc										*)
(* Desc:			writes the  tool description for				 	*)
(*             the specified tool row (d word)              *)
(* Author:	 	kbn														*)
(* Date:			30-May-2001												*)
(* Revision:	VER 4.0.0  												*)
(* last edit:	VER 6.2.33 						                  *)
(*==========================================================*)

FUNCTION_BLOCK ItpWriteToolDesc
VAR_INPUT
	bExecute:	BOOL;
	nChnId:		UDINT;
	nDNo:			UDINT;
	tTimeOut:	TIME := DEFAULT_ADS_TIMEOUT;
END_VAR
VAR_IN_OUT
	sToolDesc:	ToolDesc;
END_VAR
VAR_OUTPUT
	bBusy:		BOOL	:= FALSE;
	bErr:			BOOL	:= FALSE;
	nErrId:		UDINT	:= 0;
END_VAR
VAR
	nState:			UDINT	:= 0;
	nOffsetDNo:		UDINT	:= 0;
	nTemp:			INT;
	fbWriteParams:	ADSWRITE;
END_VAR
VAR CONSTANT
	DNO_MIN:		UDINT	:= 1;
(*	DNO_MAX:		UDINT := 50;*)

	(* index offsets *)
	IDXOFFSET_PARAMS:	UDINT	:= 16#00040000;
END_VAR
(*
Version history:
09/22/2003    | 5.4.13     | V2.9.0 (Build 947) | kbn             | adjustable target port cf. issue #2304
              |            | saved as 2.8       |                 |
*)
CASE nState OF
0:
	IF bExecute THEN
		bBusy		:= TRUE;
		bErr		:= FALSE;
		nErrId	:= 0;

		nState	:= 10;
	END_IF

10:
	(* check nDNo *)
	IF nDNo < DNO_MIN OR nDNo > NCI_MAX_TOOLDESC THEN
		(* d number out of range *)
		bErr		:= TRUE;
		nErrId	:= ErrTcNciItp_DNo;
		nState	:= 999;
	ELSE
		nOffsetDNo	:= SHL( nDNo,  8 );

		nTemp	:= SIZEOF( sToolDesc );

		fbWriteParams(
			NETID		:= '',
			PORT		:= g_NcPortTcNci,
			IDXGRP	:= NCIDXG_CHN_PARMS + nChnId,
			IDXOFFS	:= IDXOFFSET_PARAMS + nOffsetDNo,
			LEN		:= SIZEOF( sToolDesc ),
			SRCADDR	:= ADR( sToolDesc ),
			WRITE		:= TRUE,
			TMOUT		:= tTimeOut );

		nState	:= 20;
	END_IF

20:
	(* wait until all write commands are executed *)
	fbWriteParams();

	IF NOT fbWriteParams.BUSY THEN
		IF NOT fbWriteParams.ERR THEN
			nState	:= 30;
		ELSE
			bErr		:= TRUE;
			nErrId	:= fbWriteParams.ERRID;
			nState	:= 999;
		END_IF
	END_IF
30:
	(* everthing ok and done *)
	fbWriteParams( WRITE := FALSE );

	bBusy	:= FALSE;
	IF NOT bExecute THEN
		nState	:= 0;
	END_IF

999:
	(* error handling *)
	fbWriteParams( WRITE := FALSE );

	bBusy	:= FALSE;
	IF NOT bExecute THEN
		nState	:= 0;
	END_IF

END_CASE
END_FUNCTION_BLOCK

(* POU ItpWriteToolDescEx, ST *)
(*==========================================================*)
(* Name:			ItpWriteToolDescEx						         *)
(* Desc:			writes the  tool description for				 	*)
(*             the specified tool row (d word)              *)
(* Author:	 	kbn														*)
(* Date:			26-September-2006										*)
(* last edit:	VER 6.2.33 						                  *)
(*==========================================================*)

FUNCTION_BLOCK ItpWriteToolDescEx
VAR_INPUT
	bExecute:	BOOL;
	nDNo:			UDINT;
	tTimeOut:	TIME := DEFAULT_ADS_TIMEOUT;
END_VAR
VAR_IN_OUT
	sNciToPlc:	NciChannelToPlc;
	sToolDesc:	ToolDesc;
END_VAR
VAR_OUTPUT
	bBusy:		BOOL	:= FALSE;
	bErr:			BOOL	:= FALSE;
	nErrId:		UDINT	:= 0;
END_VAR
VAR
	nState:		UDINT := 0;
	fbWriteToolDesc:	ItpWriteToolDesc;
END_VAR
CASE nState OF
0:
	IF bExecute THEN
		IF ItpGetItfVersion( sNciToPlc ) > 0 THEN
			fbWriteToolDesc(
				bExecute	:= TRUE,
				nChnId	:= ItpGetChannelId( sNciToPlc ),
				nDNo		:= nDNo,
				tTimeOut	:= tTimeOut,
				sToolDesc:= sToolDesc,
				bBusy	=> bBusy,
				bErr	=> bErr,
				nErrId=> nErrId );
			nState	:= 10;
		ELSE
			bBusy		:= TRUE;
			bErr		:= TRUE;
			nErrId	:= ErrTcNciItp_ItfVersion;
			nState	:= 9999;
		END_IF
	END_IF
10:
	fbWriteToolDesc( sToolDesc := sToolDesc );
	IF NOT fbWriteToolDesc.bBusy THEN
		bBusy	:= FALSE;
		IF NOT fbWriteToolDesc.bErr THEN
			IF NOT bExecute THEN
				fbWriteToolDesc( bExecute:=FALSE, sToolDesc:=sToolDesc );
				nState	:= 0;
			ELSE
				nState	:= 9999;
			END_IF
		ELSE
			bErr		:= TRUE;
			nErrId	:= fbWriteToolDesc.nErrId;
			nState	:= 9999;
		END_IF
	END_IF

9999:
	fbWriteToolDesc( bExecute:=FALSE, sToolDesc:=sToolDesc );
	bBusy	:= FALSE;
	IF NOT bExecute THEN
		nState	:= 0;
	END_IF

END_CASE
END_FUNCTION_BLOCK

(* POU ItpWriteZeroShift, ST *)
(* Name:			ItpWriteZeroShift										*)
(* Desc:			writes the zero shift values of 					*)
(*             the specified zero shift number              *)
(* Author:	 	kbn														*)
(* Date:			30-May-2001												*)
(* Revision:	VER 4.0.0  												*)
(* last edit:	VER 6.2.33 						                  *)
(*==========================================================*)

FUNCTION_BLOCK ItpWriteZeroShift
VAR_INPUT
	bExecute:	BOOL;
	nChnId:		UDINT;
	nZsNo:		UDINT;
	tTimeOut:	TIME := DEFAULT_ADS_TIMEOUT;
END_VAR
VAR_IN_OUT
	sZeroShiftDesc:	ZeroShiftDesc;
END_VAR
VAR_OUTPUT
	bBusy:		BOOL	:= FALSE;
	bErr:			BOOL	:= FALSE;
	nErrId:		UDINT	:= 0;
END_VAR
VAR
	nState:			UDINT	:= 0;
	fShiftX:			LREAL	:= 0.0;
	fShiftY:			LREAL	:= 0.0;
	fShiftZ:			LREAL	:= 0.0;
	fbAdsWriteX:	ADSWRITE;
	fbAdsWriteY:	ADSWRITE;
	fbAdsWriteZ:	ADSWRITE;
END_VAR
VAR CONSTANT
	ZSNO_MIN:		UDINT	:= 54;
	ZSNOADJ_MAX:	UDINT := 57;

	NCIDXO_CHNP_ITPZS:	UDINT	:= 16#00010000;
	ZeroShiftX:				UDINT	:= 16#00000100;
	ZeroShiftY:				UDINT	:= 16#00000200;
	ZeroShiftZ:				UDINT	:= 16#00000300;
END_VAR
(*
Version history:
09/22/2003    | 5.4.13     | V2.9.0 (Build 947) | kbn             | adjustable target port cf. issue #2304
              |            | saved as 2.8       |                 |
*)
CASE nState OF
0:
	IF bExecute THEN
		bBusy		:= TRUE;
		bErr		:= FALSE;
		nErrId	:= 0;

		nState	:= 10;
	END_IF

10:
	(* check zero shift number *)
	IF ( nZsNo < ZSNO_MIN ) OR ( nZsNo > ZSNOADJ_MAX ) THEN
		(* error *)
		bErr		:= TRUE;
		nErrId	:= ErrTcNciItp_ZeroShiftNo;
		nState	:= 999;
	ELSE
		(* IndexOffset	0x00010K0L
							K: index of axis X=1, Y=2, Z=3
							L: zero shift number
								G54F (fine)	= 1
							 	G54G (raw) 	= 2
								G55F (fine) = 3 ...
		*)

		(* write zero shift fine *)
		fbAdsWriteX(
			NETID		:= '',
			PORT		:= g_NcPortTcNci,
			IDXGRP	:= NCIDXG_CHN_PARMS + nChnId,
			IDXOFFS	:= NCIDXO_CHNP_ITPZS + ZeroShiftX + (nZsNo - ZSNO_MIN)*2 + 1,
			LEN		:= SIZEOF( sZeroShiftDesc.fShiftX ),
			SRCADDR	:= ADR( sZeroShiftDesc.fShiftX ),
			WRITE		:= TRUE,
			TMOUT		:= tTimeOut);

		fbAdsWriteY(
			NETID		:= '',
			PORT		:= g_NcPortTcNci,
			IDXGRP	:= NCIDXG_CHN_PARMS + nChnId,
			IDXOFFS	:= NCIDXO_CHNP_ITPZS + ZeroShiftY + (nZsNo - ZSNO_MIN)*2 + 1,
			LEN		:= SIZEOF( sZeroShiftDesc.fShiftY ),
			SRCADDR	:= ADR( sZeroShiftDesc.fShiftY ),
			WRITE		:= TRUE,
			TMOUT		:= tTimeOut);

		fbAdsWriteZ(
			NETID		:= '',
			PORT		:= g_NcPortTcNci,
			IDXGRP	:= NCIDXG_CHN_PARMS + nChnId,
			IDXOFFS	:= NCIDXO_CHNP_ITPZS + ZeroShiftZ + (nZsNo - ZSNO_MIN)*2 + 1,
			LEN		:= SIZEOF( sZeroShiftDesc.fShiftZ ),
			SRCADDR	:= ADR( sZeroShiftDesc.fShiftZ ),
			WRITE		:= TRUE,
			TMOUT		:= tTimeOut);

		nState	:= 20;
	END_IF

20:
	(* wait until values are written *)
	fbAdsWriteX();
	fbAdsWriteY();
	fbAdsWriteZ();

	IF fbAdsWriteX.ERR THEN
		bErr		:= TRUE;
		nErrId	:= fbAdsWriteX.ERRID;
		nState	:= 999;
	END_IF

	IF fbAdsWriteY.ERR AND NOT bERR THEN
		bErr		:= TRUE;
		nErrId	:= fbAdsWriteY.ERRID;
		nState	:= 999;
	END_IF

	IF fbAdsWriteZ.ERR AND NOT bERR THEN
		bErr		:= TRUE;
		nErrId	:= fbAdsWriteZ.ERRID;
		nState	:= 999;
	END_IF

	IF ( NOT fbAdsWriteX.BUSY ) AND ( NOT fbAdsWriteY.BUSY ) AND ( NOT fbAdsWriteZ.BUSY ) THEN
		IF NOT bERR THEN
			nState	:= 30;
		END_IF
	END_IF

30:
	fbAdsWriteX( WRITE := FALSE );
	fbAdsWriteY( WRITE := FALSE );
	fbAdsWriteZ( WRITE := FALSE );

	nState	:= 40;

40:
	(* set raw zero shifts to zero *)
	fbAdsWriteX(
		NETID		:= '',
		PORT		:= g_NcPortTcNci,
		IDXGRP	:= NCIDXG_CHN_PARMS + nChnId,
		IDXOFFS	:= NCIDXO_CHNP_ITPZS + ZeroShiftX + (nZsNo - ZSNO_MIN)*2 + 2,
		LEN		:= SIZEOF( fShiftX ),
		SRCADDR	:= ADR( fShiftX ),
		WRITE		:= TRUE,
		TMOUT		:= tTimeOut);

	fbAdsWriteY(
		NETID		:= '',
		PORT		:= g_NcPortTcNci,
		IDXGRP	:= NCIDXG_CHN_PARMS + nChnId,
		IDXOFFS	:= NCIDXO_CHNP_ITPZS + ZeroShiftY + (nZsNo - ZSNO_MIN)*2 + 2,
		LEN		:= SIZEOF( fShiftY ),
		SRCADDR	:= ADR( fShiftY ),
		WRITE		:= TRUE,
		TMOUT		:= tTimeOut);

	fbAdsWriteZ(
		NETID		:= '',
		PORT		:= g_NcPortTcNci,
		IDXGRP	:= NCIDXG_CHN_PARMS + nChnId,
		IDXOFFS	:= NCIDXO_CHNP_ITPZS + ZeroShiftZ + (nZsNo - ZSNO_MIN)*2 + 2,
		LEN		:= SIZEOF( fShiftZ ),
		SRCADDR	:= ADR( fShiftZ ),
		WRITE		:= TRUE,
		TMOUT		:= tTimeOut);

	nState	:= 50;

50:
	(* wait until raw values are written *)
	fbAdsWriteX();
	fbAdsWriteY();
	fbAdsWriteZ();

	IF fbAdsWriteX.ERR THEN
		bErr		:= TRUE;
		nErrId	:= fbAdsWriteX.ERRID;
		nState	:= 999;
	END_IF

	IF fbAdsWriteY.ERR AND NOT bERR THEN
		bErr		:= TRUE;
		nErrId	:= fbAdsWriteY.ERRID;
		nState	:= 999;
	END_IF

	IF fbAdsWriteZ.ERR AND NOT bERR THEN
		bErr		:= TRUE;
		nErrId	:= fbAdsWriteZ.ERRID;
		nState	:= 999;
	END_IF

	IF ( NOT fbAdsWriteX.BUSY ) AND ( NOT fbAdsWriteY.BUSY ) AND ( NOT fbAdsWriteZ.BUSY ) THEN
		IF NOT bERR THEN
			nState	:= 60;
		END_IF
	END_IF

60:
	(* everthing is ok & done *)
	fbAdsWriteX( WRITE := FALSE );
	fbAdsWriteY( WRITE := FALSE );
	fbAdsWriteZ( WRITE := FALSE );

	bBusy	:= FALSE;

	IF NOT bExecute THEN
		nState	:= 0;
	END_IF

999:
	(* error handling *)
	fbAdsWriteX( WRITE := FALSE );
	fbAdsWriteY( WRITE := FALSE );
	fbAdsWriteZ( WRITE := FALSE );

	bBusy	:= FALSE;

	IF NOT bExecute THEN
		nState	:= 0;
	END_IF

END_CASE
END_FUNCTION_BLOCK

(* POU ItpWriteZeroShiftEx, ST *)
(*==========================================================*)
(* Name:			ItpWriteZeroShiftEx						         *)
(* Desc:			writes the zero shift values of 					*)
(*             the specified zero shift number              *)
(* Author:	 	kbn														*)
(* Date:			26-September-2006										*)
(* last edit:	VER 6.2.33 						                  *)
(*==========================================================*)

FUNCTION_BLOCK ItpWriteZeroShiftEx
VAR_INPUT
	bExecute:	BOOL;
	nZsNo:		UDINT;
	tTimeOut:	TIME := DEFAULT_ADS_TIMEOUT;
END_VAR
VAR_IN_OUT
	sNciToPlc:			NciChannelToPlc;
	sZeroShiftDesc:	ZeroShiftDesc;
END_VAR
VAR_OUTPUT
	bBusy:		BOOL	:= FALSE;
	bErr:			BOOL	:= FALSE;
	nErrId:		UDINT	:= 0;
END_VAR
VAR
	nState:		UDINT := 0;
	fbItpWriteZeroShift:	ItpWriteZeroShift;
END_VAR
CASE nState OF
0:
	IF bExecute THEN
		IF ItpGetItfVersion( sNciToPlc ) > 0 THEN
			fbItpWriteZeroShift(
				bExecute	:= TRUE,
				nChnId	:= ItpGetChannelId( sNciToPlc ),
				nZsNo		:= nZsNo,
				tTimeOut	:= tTimeOut,
				sZeroShiftDesc:= sZeroShiftDesc,
				bBusy	=> bBusy,
				bErr	=> bErr,
				nErrId=> nErrId );
			nState	:= 10;
		ELSE
			bBusy		:= TRUE;
			bErr		:= TRUE;
			nErrId	:= ErrTcNciItp_ItfVersion;
			nState	:= 9999;
		END_IF
	END_IF
10:
	fbItpWriteZeroShift( sZeroShiftDesc := sZeroShiftDesc );
	IF NOT fbItpWriteZeroShift.bBusy THEN
		bBusy	:= FALSE;
		IF NOT fbItpWriteZeroShift.bErr THEN
			IF NOT bExecute THEN
				fbItpWriteZeroShift( bExecute:=FALSE, sZeroShiftDesc:=sZeroShiftDesc );
				nState	:= 0;
			ELSE
				nState	:= 9999;
			END_IF
		ELSE
			bErr		:= TRUE;
			nErrId	:= fbItpWriteZeroShift.nErrId;
			nState	:= 9999;
		END_IF
	END_IF

9999:
	fbItpWriteZeroShift( bExecute:=FALSE, sZeroShiftDesc:=sZeroShiftDesc );
	bBusy	:= FALSE;
	IF NOT bExecute THEN
		nState	:= 0;
	END_IF

END_CASE
END_FUNCTION_BLOCK
